{attribute 'qualified_only'}
VAR_GLOBAL
	//Test
	{attribute 'OPC.UA.DA' := '1'}
	reactorTemperatureContactor AT %Q* : BOOL; // Temperature contactor
	reactorTemperatureUpper AT %I*: INT; // Reactor temperature
	reactorTemperatureLower AT %I*: INT; // Reactor temperature lower
	reactorLevelHigherHigh AT %I*: BOOL; // Higher high slurry level
	reactorLevelHigh AT %I*: BOOL; // High slurry level
	reactorLevelLower AT %I*: BOOL; // Low slurry level
	reactorLevelLowerLow AT %I*: BOOL; // Lower low slurry level
	reactorOutletValve AT %Q*: BOOL;  // Reactor outlet valve
	reactorPressure AT %I*: INT; // Reactor pressure raw analog value
	reactorInletValve AT %Q*: BOOL; // Filling valve
END_VAR

(* stored: Version 1.1.0.1, ProductVersion 3.1.4024.9
   GVL IO: Id {86a3f261-87c7-445b-99f5-4f998ed6afb1} *)
